TYPE IO_typ:
STRUCT
	EL1008: EL1008IO_typ;
	EL2008: EL2008IO_typ;
END_STRUCT
END_TYPE

(* stored: Version 1.1.0.1, ProductVersion 3.1.4024.12
   DUT IO_typ: Id {ea205016-8f1b-0d1c-2b29-aead27e63e0a} *)
